FUNCTION_BLOCK EL3141
VAR
	_io : EL3xx1_Data;
	{attribute addProperty Name "WcState"}
	_wcState : WcStateInputToggle;
	{attribute addProperty Name "Info data"}
	_infoData : InfoDataAds;
END_VAR

PROPERTY IO : REFERENCE TO EL3xx1_Data
GET
IO REF= _io;
END_GET
END_PROPERTY

PROPERTY WcState : REFERENCE TO WcStateInputToggle
GET
WcState REF= _wcState;
END_GET
END_PROPERTY

END_FUNCTION_BLOCK

(* stored: Version 1.1.0.1, ProductVersion 3.1.4024.9
   POU EL3141: Id {e33bf73f-9dd0-08c0-098e-4829edb11276}, SpecialFunc None
   Property IO: Id {3bc9e99e-ba95-0680-1d68-74a91b8e46e0}
   Get Get: Id {a43e6717-f4ec-0f3a-2838-b5155acbf92b}
   Property WcState: Id {0bbe2865-ba88-0220-0853-6091fe71afc9}
   Get Get: Id {61afbdf4-a740-04d2-1f4b-4c00d5e652b0} *)
